// TIA Portal V20 export
// export: Created 2025-12-01T14:56:17.650015Z, ExportSetting None, DisplayName Totally Integrated Automation Portal, DisplayVersion V20 Update 3, DisplayName TIA Portal Openness, DisplayVersion V20 Update 3, DisplayName TIA Portal Version Control Interface, DisplayVersion V20 Update 3, DisplayName STEP 7 Professional, DisplayVersion V20 Update 3, DisplayName STEP 7 Safety, DisplayVersion V20 Update 2, DisplayName WinCC Basic/Comfort/Advanced, DisplayVersion V20 Update 3, DisplayName WinCC Professional, DisplayVersion V20 Update 3, DisplayName WinCC Unified, DisplayVersion V20 Update 3
TYPE "UDT_ScadaDatosMesa"
   STRUCT
      Ordenes_S0 : Bool;
      Ordenes_S1 : Bool;
      Ordenes_S2 : Bool;
      Ordenes_S3 : Bool;
      Ordenes_S4 : Bool;
      Libre_05 : Bool;
      Libre_06 : Bool;
      Libre_07 : Bool;
      Aviso_E1 : Bool;
      Permiso_E1 : Bool;
      Fin_E1 : Bool;
      Aviso_E2 : Bool;
      Permiso_E2 : Bool;
      Fin_E2 : Bool;
      Aviso_E3 : Bool;
      Permiso_E3 : Bool;
      Fin_E3 : Bool;
      Aviso_E4 : Bool;
      Permiso_E4 : Bool;
      Fin_E4 : Bool;
      Aviso_S1 : Bool;
      Permiso_S1 : Bool;
      Fin_S1 : Bool;
      Aviso_S2 : Bool;
      Permiso_S2 : Bool;
      Fin_S2 : Bool;
      Aviso_S3 : Bool;
      Permiso_S3 : Bool;
      Fin_S3 : Bool;
      Aviso_S4 : Bool;
      Permiso_S4 : Bool;
      Fin_S4 : Bool;
      Bultos_Totales : UInt;
      Bultos_E1 : UInt;
      Bultos_E2 : UInt;
      Bultos_E3 : UInt;
      Bultos_E4 : UInt;
      Bultos_S1 : UInt;
      Bultos_S2 : UInt;
      Bultos_S3 : UInt;
      Bultos_S4 : UInt;
      TMP_Error : Time_Of_Day;
      Arranques_M1 : UInt;   // M1 -> Motor Principal
      TMP_Marcha_M1 : Time_Of_Day;
      Arranques_M2 : UInt;   // M2 -> Motor Secundario
      TMP_Marcha_M2 : Time_Of_Day;
      Arranques_M3 : UInt;   // M3 -> Motor Giro
      TMP_Marcha_M3 : Time_Of_Day;
      Arranques_M4 : UInt;   // M4 -> Motor de Elevacion
      TMP_Marcha_M4 : Time_Of_Day;
      Arranques_M5 : UInt;   // M5 -> Motor de Tope
      TMP_Marcha_M5 : Time_Of_Day;
      MemoBultos_Totales : Bool;
      MemoBultos_E1 : Bool;
      MemoBultos_E2 : Bool;
      MemoBultos_E3 : Bool;
      MemoBultos_E4 : Bool;
      MemoBultos_S1 : Bool;
      MemoBultos_S2 : Bool;
      MemoBultos_S3 : Bool;
      MemoBultos_S4 : Bool;
      MemoArranques_M1 : Bool;   // M1 -> Motor Principal
      MemoArranques_M2 : Bool;   // M2 -> Motor Secundario
      MemoArranques_M3 : Bool;   // M3 -> Motor Giro
      MemoArranques_M4 : Bool;   // M4 -> Motor de Elevacion
      MemoArranques_M5 : Bool;   // M5 -> Motor de Tope
      Libre_576 : Bool;
      Libre_577 : Bool;
   END_STRUCT;
END_TYPE
